	28:
		tbTBLog := CONCAT(tbTBLog, INT_TO_STRING(iTestStep));
		FOR i := 1 TO 3 DO
			IF gaTemps[i].stDescription.xFault = TRUE OR gaTemps[i].stDescription.xAlarm = TRUE THEN
				tbTBLog := CONCAT(tbTBLog, 'F');
				iTestStep := 66;
			ELSE
				tbTBLog := CONCAT(tbTBLog, 'S');
				iTestStep := iTestStep + 1;
			END_IF
		END_FOR
	29:
		tbTBLog := CONCAT(tbTBLog, INT_TO_STRING(iTestStep));
		IF gConductivity.stDescription.xFault = FALSE OR gConductivity.stDescription.xAlarm = FALSE THEN
				tbTBLog := CONCAT(tbTBLog, 'F');
				iTestStep := 66;
		ELSE
				tbTBLog := CONCAT(tbTBLog, 'S');
				iTestStep := iTestStep + 1;
		END_IF
	30:
		tbTBLog := CONCAT(tbTBLog, INT_TO_STRING(iTestStep));
		IF gFlow.stDescription.xFault = TRUE OR gFlow.stDescription.xAlarm = TRUE THEN
				tbTBLog := CONCAT(tbTBLog, 'F ');
				iTestStep := 66;
		ELSE
				tbTBLog := CONCAT(tbTBLog, 'S');
				iTestStep := iTestStep + 1;
		END_IF
	31: (*Max Val Test Cond Should Fault*)
		resetVars();
		tbTBLog := CONCAT(tbTBLog, INT_TO_STRING(iTestStep));
		gaPumps[1].stPumpPower.iRaw := 5;
		gaPumps[2].stPumpPower.iRaw := 5;
		gaTemps[i].stTempRead.iRaw := 5;
		gaTemps[2].stTempRead.iRaw := 5;
		gaTemps[3].stTempRead.iRaw := 5;
		gConductivity.stConductivity.iRaw := 100;
		gFlow.stFlowRate.iRaw := 5;
		UUT();
		tbTBLog := CONCAT(tbTBLog, 'S');
		iTestStep := iTestStep + 1;
	32:
		tbTBLog := CONCAT(tbTBLog, INT_TO_STRING(iTestStep));
		FOR i := 1 TO 2 DO
			IF gaPumps[i].stDescription.xFault = TRUE OR gaPumps[i].stDescription.xAlarm = TRUE THEN
				tbTBLog := CONCAT(tbTBLog, 'F');
				iTestStep := 66;
			ELSE
				tbTBLog := CONCAT(tbTBLog, 'S');
				iTestStep := iTestStep + 1;
			END_IF
		END_FOR

	33:
		tbTBLog := CONCAT(tbTBLog, INT_TO_STRING(iTestStep));
		FOR i := 1 TO 3 DO
			IF gaTemps[i].stDescription.xFault = TRUE OR gaTemps[i].stDescription.xAlarm = TRUE THEN
				tbTBLog := CONCAT(tbTBLog, 'F');
				iTestStep := 66;
			ELSE
				tbTBLog := CONCAT(tbTBLog, 'S');
				iTestStep := iTestStep + 1;
			END_IF
		END_FOR
	34:
		tbTBLog := CONCAT(tbTBLog, INT_TO_STRING(iTestStep));
		IF gConductivity.stDescription.xFault = FALSE OR gConductivity.stDescription.xAlarm = FALSE THEN
				tbTBLog := CONCAT(tbTBLog, 'F');
				iTestStep := 66;
		ELSE
				tbTBLog := CONCAT(tbTBLog, 'S');
				iTestStep := iTestStep + 1;
		END_IF
	35:
		tbTBLog := CONCAT(tbTBLog, INT_TO_STRING(iTestStep));
		IF gFlow.stDescription.xFault = TRUE OR gFlow.stDescription.xAlarm = TRUE THEN
				tbTBLog := CONCAT(tbTBLog, 'F ');
				iTestStep := 66;
		ELSE
				tbTBLog := CONCAT(tbTBLog, 'S');
				iTestStep := iTestStep + 1;
		END_IF
	36: (*MIN Val Test Flow Should Fault*)
		resetVars();
		tbTBLog := CONCAT(tbTBLog, INT_TO_STRING(iTestStep));
		gaPumps[1].stPumpPower.iRaw := 5;
		gaPumps[2].stPumpPower.iRaw := 5;
		gaTemps[i].stTempRead.iRaw := 5;
		gaTemps[2].stTempRead.iRaw := 5;
		gaTemps[3].stTempRead.iRaw := 5;
		gConductivity.stConductivity.iRaw := 5;
		gFlow.stFlowRate.iRaw := 1;
		UUT();
		tbTBLog := CONCAT(tbTBLog, 'S');
		iTestStep := iTestStep + 1;
	37:
		tbTBLog := CONCAT(tbTBLog, INT_TO_STRING(iTestStep));
		FOR i := 1 TO 2 DO
			IF gaPumps[i].stDescription.xFault = TRUE OR gaPumps[i].stDescription.xAlarm = TRUE THEN
				tbTBLog := CONCAT(tbTBLog, 'F');
				iTestStep := 66;
			ELSE
				tbTBLog := CONCAT(tbTBLog, 'S');
				iTestStep := iTestStep + 1;
			END_IF
		END_FOR

	38:
		tbTBLog := CONCAT(tbTBLog, INT_TO_STRING(iTestStep));
		FOR i := 1 TO 3 DO
			IF gaTemps[i].stDescription.xFault = TRUE OR gaTemps[i].stDescription.xAlarm = TRUE THEN
				tbTBLog := CONCAT(tbTBLog, 'F');
				iTestStep := 66;
			ELSE
				tbTBLog := CONCAT(tbTBLog, 'S');
				iTestStep := iTestStep + 1;
			END_IF
		END_FOR
	39:
		tbTBLog := CONCAT(tbTBLog, INT_TO_STRING(iTestStep));
		IF gConductivity.stDescription.xFault = TRUE OR gConductivity.stDescription.xAlarm = TRUE THEN
				tbTBLog := CONCAT(tbTBLog, 'F');
				iTestStep := 66;
		ELSE
				tbTBLog := CONCAT(tbTBLog, 'S');
				iTestStep := iTestStep + 1;
		END_IF
	40:
		tbTBLog := CONCAT(tbTBLog, INT_TO_STRING(iTestStep));
		IF gFlow.stDescription.xFault = FALSE  OR gFlow.stDescription.xAlarm = FALSE THEN
				tbTBLog := CONCAT(tbTBLog, 'F ');
				iTestStep := 66;
		ELSE
				tbTBLog := CONCAT(tbTBLog, 'S');
				iTestStep := iTestStep + 1;
		END_IF
	41: (*MAX Val Test Flow Should Fault*)
		resetVars();
		tbTBLog := CONCAT(tbTBLog, INT_TO_STRING(iTestStep));
		gaPumps[1].stPumpPower.iRaw := 5;
		gaPumps[2].stPumpPower.iRaw := 5;
		gaTemps[i].stTempRead.iRaw := 5;
		gaTemps[2].stTempRead.iRaw := 5;
		gaTemps[3].stTempRead.iRaw := 5;
		gConductivity.stConductivity.iRaw := 5;
		gFlow.stFlowRate.iRaw := 100;
		UUT();
		tbTBLog := CONCAT(tbTBLog, 'S');
		iTestStep := iTestStep + 1;
	42:
		tbTBLog := CONCAT(tbTBLog, INT_TO_STRING(iTestStep));
		FOR i := 1 TO 2 DO
			IF gaPumps[i].stDescription.xFault = TRUE OR gaPumps[i].stDescription.xAlarm = TRUE THEN
				tbTBLog := CONCAT(tbTBLog, 'F');
				iTestStep := 66;
			ELSE
				tbTBLog := CONCAT(tbTBLog, 'S');
				iTestStep := iTestStep + 1;
			END_IF
		END_FOR

	43:
		tbTBLog := CONCAT(tbTBLog, INT_TO_STRING(iTestStep));
		FOR i := 1 TO 3 DO
			IF gaTemps[i].stDescription.xFault = TRUE OR gaTemps[i].stDescription.xAlarm = TRUE THEN
				tbTBLog := CONCAT(tbTBLog, 'F');
				iTestStep := 66;
			ELSE
				tbTBLog := CONCAT(tbTBLog, 'S');
				iTestStep := iTestStep + 1;
			END_IF
		END_FOR
	44:
		tbTBLog := CONCAT(tbTBLog, INT_TO_STRING(iTestStep));
		IF gConductivity.stDescription.xFault = TRUE OR gConductivity.stDescription.xAlarm = TRUE THEN
				tbTBLog := CONCAT(tbTBLog, 'F');
				iTestStep := 66;
		ELSE
				tbTBLog := CONCAT(tbTBLog, 'S');
				iTestStep := iTestStep + 1;
		END_IF
	45:
		tbTBLog := CONCAT(tbTBLog, INT_TO_STRING(iTestStep));
		IF gFlow.stDescription.xFault = FALSE  OR gFlow.stDescription.xAlarm = FALSE THEN
				tbTBLog := CONCAT(tbTBLog, 'F ');
				iTestStep := 66;
		ELSE
				tbTBLog := CONCAT(tbTBLog, 'S');
				iTestStep := iTestStep + 1;
		END_IF
END_CASE
*)
END_PROGRAM

(* POU Legacy/FB_TempValCtrlSys, ST *)
FUNCTION_BLOCK FB_TempValCtrlSys
VAR_INPUT
END_VAR
VAR_OUTPUT
END_VAR
VAR
	tM: ARRAY [1..3] OF REAL; (*Temperature Measuremnts*)
	tD: ARRAY [1..3] OF REAL; (*Temperature differences of 1 and 2, 1 and 3, 2 and 3*)
	tCF: ARRAY [1..3] OF BOOL; (*Candiates of potential temperatures that failed. First true means 1 and 2. Second true means 1 and 3. And third true means 2 and 3.*)
	tCA: ARRAY [1..3] OF BOOL; (*Candiates of potential temperatures that alarmed. First true means 1 and 2. Second true means 1 and 3. And third true means 2 and 3.*)

	i: INT;
	diffThreshold: REAL;
	diffTolerance: REAL;
	faultCount: INT; (*How many faults*)
	sysMeasMode: INT;
END_VAR
faultCount := 0;
i := 0;
(*Subtract to find differneces between temperatures*)
FOR i := 1 TO 3 DO
	tM[i] := gaTemps[i].stTempRead.rProcessed;
END_FOR
tD[1] := ABS(tM[1] - tM[2]);
tD[2] := ABS(tM[1] - tM[3]);
tD[3] := ABS(tM[2] - tM[3]);
i := 0;
FOR i := 1 TO 3 DO
	IF tD[i] > gTempValCtrlSys.rDiffThresh THEN
		tCF[i] := TRUE;
		tCA[i] := TRUE;
		faultCount := faultCount + 1;
		gTempValCtrlSys.xAlarm := TRUE;
	ELSIF tD[i] > (gTempValCtrlSys.rDiffTol) THEN
		tCA[i] := TRUE;
		gTempValCtrlSys.xAlarm := TRUE;
END_IF
END_FOR
IF tCF[1] = TRUE AND tCF[2] = TRUE AND tCF[3] = TRUE THEN
	FOR i := 1 TO 3 DO
		gaTemps[i].stDescription.xFault := TRUE;
	END_FOR
ELSIF tCF[1] = TRUE AND tCF[2] = TRUE AND tCF[3] = FALSE THEN
	gaTemps[1].stDescription.xFault := TRUE;
ELSIF tCF[1] = TRUE AND tCF[2] = FALSE AND tCF[3] = TRUE THEN
	gaTemps[2].stDescription.xFault := TRUE;
ELSIF tCF[1] = FALSE AND tCF[2] = TRUE AND tCF[3] = TRUE THEN
	gaTemps[3].stDescription.xFault := TRUE;

END_IF

IF tCA[1] = TRUE AND tCA[2] = TRUE AND tCA[3] = TRUE THEN
	FOR i := 1 TO 3 DO
		gaTemps[i].stDescription.xAlarm:= TRUE;
	END_FOR
ELSIF tCA[1] = TRUE AND tCA[2] = TRUE AND tCA[3] = FALSE THEN
	gaTemps[1].stDescription.xAlarm := TRUE;
ELSIF tCA[1] = TRUE AND tCA[2] = FALSE AND tCA[3] = TRUE THEN
	gaTemps[2].stDescription.xAlarm := TRUE;
ELSIF tCA[1] = FALSE AND tCA[2] = TRUE AND tCA[3] = TRUE THEN
	gaTemps[3].stDescription.xAlarm := TRUE;
END_IF

IF faultCount = 0 THEN
	sysMeasMode := 0;
ELSIF faultCount = 1 THEN
	gProgramErrors.xTempValCtrlSys  := TRUE; (*If difference between only two RTDs off, means poor values selected*)
	gTempValCtrlSys.xFault := TRUE;
	gTempValCtrlSys.xAlarm := TRUE;
ELSIF faultCount = 2 THEN (*Means that an RTD failed, will need to take average *)
	sysMeasMode := 1;
	gTempValCtrlSys.xAlarm := TRUE;
ELSIF faultCount = 3 THEN (*All RTDs failed, system fault*)
	sysMeasMode := 2;
	gTempValCtrlSys.xFault := TRUE;
	gTempValCtrlSys.xAlarm := TRUE;
ELSE (*Should not happen*)
	gProgramErrors.xTempValCtrlSys  := TRUE;
	gTempValCtrlSys.xFault := TRUE;
	gTempValCtrlSys.xAlarm := TRUE;
END_IF
END_FUNCTION_BLOCK

(* POU Test Bench Folder/TB_VALIDATE, LD *)
PROGRAM TB_VALIDATE
VAR
	rResult: REAL;
	rinput: REAL;
	rMax: REAL;
	rMin: REAL;
	Val1: REAL;
	Val2: REAL;
	Val3: REAL;
	bool1: BOOL := TRUE;
	bool2: BOOL := TRUE;
	bool3: BOOL := TRUE;
END_VAR
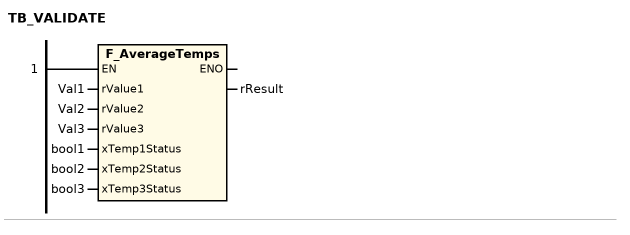
_LD_ (* Ladder Diagram *)
NETWORK 1
	*
		EN --- F_AverageTemps(rValue1: Val1, rValue2: Val2, rValue3: Val3, xTemp1Status: bool1, xTemp2Status: bool2, xTemp3Status: bool3) => rResult
_END_LD_
(* the same logic as Structured Text *)
(* Network 1 *)
rResult := F_AverageTemps(rValue1 := Val1, rValue2 := Val2, rValue3 := Val3, xTemp1Status := bool1, xTemp2Status := bool2, xTemp3Status := bool3);
END_PROGRAM

(* POU Test Bench Folder/TB_WaterLevelCheck, LD *)
PROGRAM TB_WaterLevelCheck
VAR
	fbcwl: FB_CheckWaterLevel;
	sys: ST_SYSTEM;
	wl: BOOL := FALSE;
	wll: BOOL := FALSE;
	flags: ST_InstrumentFlags;
END_VAR
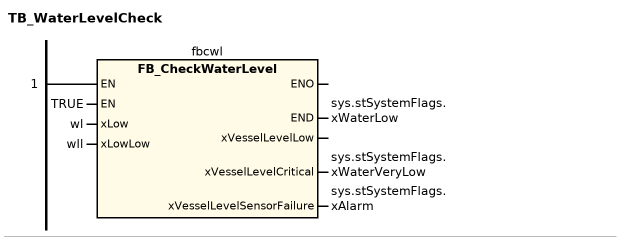
_LD_ (* Ladder Diagram *)
NETWORK 1
	*
		EN --- fbcwl:FB_CheckWaterLevel(EN: TRUE, xLow: wl, xLowLow: wll, xVesselLevelCritical => sys.stSystemFlags.xWaterVeryLow, xVesselLevelSensorFailure => sys.stSystemFlags.xAlarm) => sys.stSystemFlags.xWaterLow
_END_LD_
(* the same logic as Structured Text *)
(* Network 1 *)
fbcwl(EN := TRUE, xLow := wl, xLowLow := wll);
sys.stSystemFlags.xWaterVeryLow := fbcwl.xVesselLevelCritical;
sys.stSystemFlags.xAlarm := fbcwl.xVesselLevelSensorFailure;
sys.stSystemFlags.xWaterLow := fbcwl.END;
END_PROGRAM

(* POU System Startup/F_InitSystemCheck, ST *)
FUNCTION F_InitSystemCheck : BOOL
VAR_INPUT
	xSystemRunSwitch: BOOL;
	xSystemFaultFlag: BOOL;
END_VAR
VAR
END_VAR
IF (xSystemRunSwitch AND xSystemFaultFlag) OR (xSystemRunSwitch = FALSE) THEN
	F_InitSystemCheck := FALSE;
ELSIF xSystemRunSwitch AND xSystemFaultFlag = FALSE THEN
	F_InitSystemCheck := TRUE;
END_IF;
END_FUNCTION

(* POU Instrument Control/F_SystemFaultCheck, LD *)
FUNCTION_BLOCK F_SystemFaultCheck
VAR_INPUT
	xRTD1: BOOL;
	xRTD2: BOOL;
	xRTD3: BOOL;
	xPump1: BOOL;
	xBadWaterLevelSensor: BOOL;
	xBadConductivitySensor: BOOL;
	xBadFlowSensor: BOOL;
	xBadTemperature: BOOL;
	xLowPressure: BOOL;
	xLowFLow: BOOL;
	xNoBackup: BOOL;
	iActivePump: INT;
	xBadActuate: BOOL;
	xSystemPump1Activate: BOOL;
	xSystemPump2Activate: BOOL;
END_VAR
VAR_OUTPUT
	xSystemFault: BOOL;
END_VAR
VAR
	xBadTemp12: BOOL;
	xBadTemp23: BOOL;
	xBadTemp31: BOOL;
	xPump2: BOOL;
	xNoPump: BOOL;
	xTri1: BOOL;
	xTri2: BOOL;
	xTri3: BOOL;
END_VAR
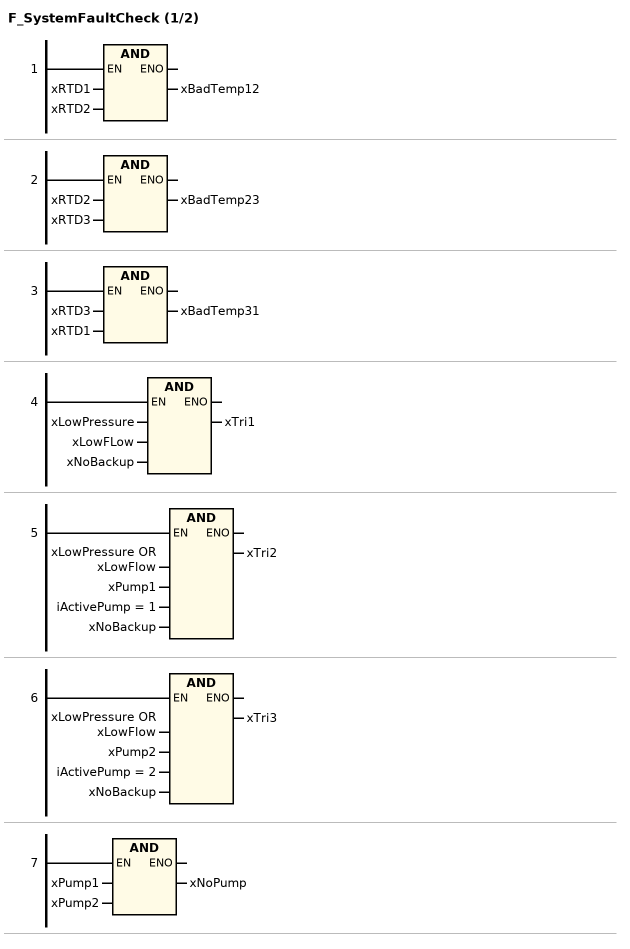
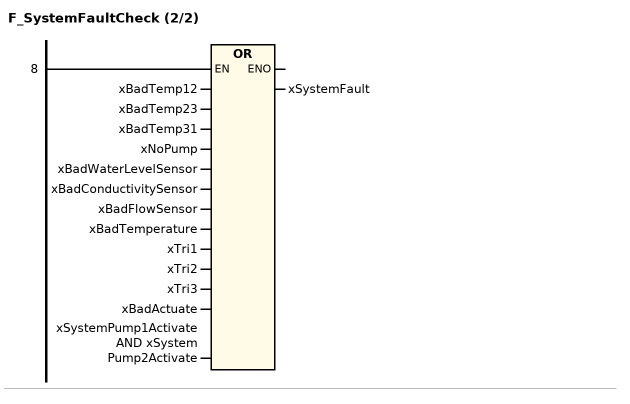
_LD_ (* Ladder Diagram *)
NETWORK 1
	*
		EN --- AND(xRTD1, xRTD2) => xBadTemp12
NETWORK 2
	*
		EN --- AND(xRTD2, xRTD3) => xBadTemp23
NETWORK 3
	*
		EN --- AND(xRTD3, xRTD1) => xBadTemp31
NETWORK 4
	*
		EN --- AND(xLowPressure, xLowFLow, xNoBackup) => xTri1
NETWORK 5
	*
		EN --- AND(xLowPressure OR xLowFlow, xPump1, iActivePump = 1, xNoBackup) => xTri2
NETWORK 6
	*
		EN --- AND(xLowPressure OR xLowFlow, xPump2, iActivePump = 2, xNoBackup) => xTri3
NETWORK 7
	*
		EN --- AND(xPump1, xPump2) => xNoPump
NETWORK 8
	*
		EN --- OR(xBadTemp12, xBadTemp23, xBadTemp31, xNoPump, xBadWaterLevelSensor, xBadConductivitySensor, xBadFlowSensor, xBadTemperature, xTri1, xTri2, xTri3, xBadActuate, xSystemPump1Activate AND xSystemPump2Activate) => xSystemFault
_END_LD_
(* the same logic as Structured Text *)
(* Network 1 *)
xBadTemp12 := xRTD1 AND xRTD2;
(* Network 2 *)
xBadTemp23 := xRTD2 AND xRTD3;
(* Network 3 *)
xBadTemp31 := xRTD3 AND xRTD1;
(* Network 4 *)
xTri1 := xLowPressure AND xLowFLow AND xNoBackup;
(* Network 5 *)
xTri2 := (xLowPressure OR xLowFlow) AND xPump1 AND (iActivePump = 1) AND xNoBackup;
(* Network 6 *)
xTri3 := (xLowPressure OR xLowFlow) AND xPump2 AND (iActivePump = 2) AND xNoBackup;
(* Network 7 *)
xNoPump := xPump1 AND xPump2;
(* Network 8 *)
xSystemFault := xBadTemp12 OR xBadTemp23 OR xBadTemp31 OR xNoPump OR xBadWaterLevelSensor OR xBadConductivitySensor OR xBadFlowSensor OR xBadTemperature OR xTri1 OR xTri2 OR xTri3 OR xBadActuate OR (xSystemPump1Activate AND xSystemPump2Activate);
END_FUNCTION_BLOCK

(* POU Instrument Control/Temperature Control/F_TemperatureController, ST *)
FUNCTION F_TemperatureController : REAL
VAR_INPUT
	xSystemFaultFlag: BOOL;
	xAwaitInit: BOOL;
	rTemperatureInput: REAL;
	rSetpoint: REAL;
END_VAR
VAR
	rOutput: REAL;
END_VAR
IF xSystemFaultFlag OR xAwaitInit THEN
	F_TemperatureController := 1;
ELSE
	F_TemperatureController :=( rTemperatureInput/2)/rTemperatureInput;
END_IF
END_FUNCTION

(* POU Functions/F_ValueCap, ST *)
FUNCTION F_ValueCap : REAL
VAR_INPUT
	rInput: REAL;
END_VAR
VAR
END_VAR
IF (rInput > 1) THEN
	F_ValueCap := 1;
ELSIF (rInput < 1) THEN
	F_ValueCap := 0;
ELSE
	F_ValueCap := rInput;
END_IF
END_FUNCTION

(* POU Data Conversion/System -> Instrument/FB_ActivePumpSet, ST *)
FUNCTION_BLOCK FB_ActivePumpSet
VAR_INPUT
	xSystemPump1Actuate: BOOL;
	xSystemPump2Actuate: BOOL;
END_VAR
VAR_OUTPUT
	iActivePump: INT;
	xSystemFaultFlag: BOOL;
END_VAR
VAR
END_VAR
IF xSystemPump1Actuate AND xSystemPump2Actuate = FALSE THEN
	iActivePump := 1;
ELSIF xSystemPump2Actuate AND xSystemPump1Actuate = FALSE THEN
	iActivePump := 2;
ELSIF xSystemPump1Actuate AND xSystemPump2Actuate THEN
	iActivePump := 0;
	xSystemFaultFlag := TRUE;
ELSIF xSystemPump1Actuate = FALSE AND xSystemPump2Actuate = FALSE THEN
	iActivePump := 0;
END_IF
END_FUNCTION_BLOCK

(* POU Data Conversion/Instrument -> Signal/FB_ActuateAnalog, LD *)
 FUNCTION_BLOCK FB_ActuateAnalog
VAR_INPUT
	rActuateValue: REAL;
END_VAR
VAR_OUTPUT
	wActuateSignal: WORD;
END_VAR
VAR
	rScaledValue: REAL;
END_VAR
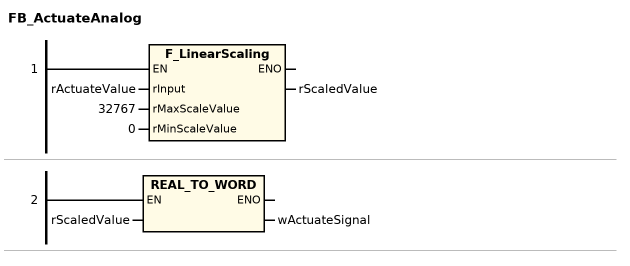
_LD_ (* Ladder Diagram *)
NETWORK 1
	*
		EN --- F_LinearScaling(rInput: rActuateValue, rMaxScaleValue: 32767, rMinScaleValue: 0) => rScaledValue
NETWORK 2
	*
		EN --- REAL_TO_WORD(rScaledValue) => wActuateSignal
_END_LD_
(* the same logic as Structured Text *)
(* Network 1 *)
rScaledValue := F_LinearScaling(rInput := rActuateValue, rMaxScaleValue := 32767, rMinScaleValue := 0);
(* Network 2 *)
wActuateSignal := REAL_TO_WORD(rScaledValue);
END_FUNCTION_BLOCK

(* POU Data Conversion/Instrument -> Signal/FB_ActuateDigital, LD *)
FUNCTION_BLOCK FB_ActuateDigital
VAR_INPUT
	xPump1ActuateValue: BOOL;
	xPump2ActuateValue: BOOL;
	xFan12ActuateValue: BOOL;
	xFan34ActuateValue: BOOL;
END_VAR
VAR_OUTPUT
	xPump1OutputSignal: BOOL;
	xPump2OutputSignal: BOOL;
	xFan12OutputSignal: BOOL;
	xFan34OutputSignal: BOOL;
END_VAR
VAR
END_VAR
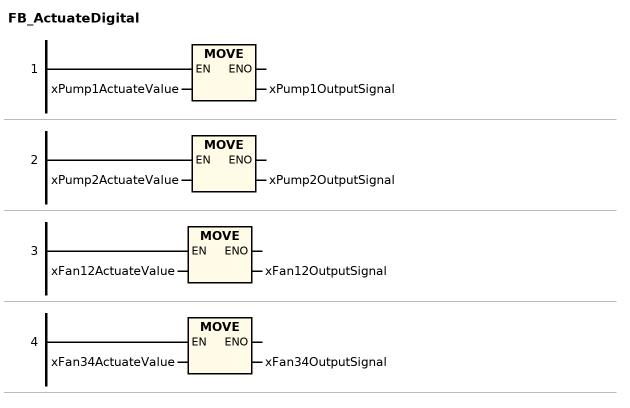
_LD_ (* Ladder Diagram *)
NETWORK 1
	*
		EN --- MOVE(xPump1ActuateValue) => xPump1OutputSignal
NETWORK 2
	*
		EN --- MOVE(xPump2ActuateValue) => xPump2OutputSignal
NETWORK 3
	*
		EN --- MOVE(xFan12ActuateValue) => xFan12OutputSignal
NETWORK 4
	*
		EN --- MOVE(xFan34ActuateValue) => xFan34OutputSignal
_END_LD_
(* the same logic as Structured Text *)
(* Network 1 *)
xPump1OutputSignal := xPump1ActuateValue;
(* Network 2 *)
xPump2OutputSignal := xPump2ActuateValue;
(* Network 3 *)
xFan12OutputSignal := xFan12ActuateValue;
(* Network 4 *)
xFan34OutputSignal := xFan34ActuateValue;
END_FUNCTION_BLOCK

(* POU Data Conversion/System -> Instrument/FB_ActuateFilter, ST *)
FUNCTION_BLOCK FB_ActuateFilter
VAR_INPUT
	rActuateValue: REAL;
	rActuateMAX: REAL;
	rActuateMIN: REAL;
END_VAR
VAR_OUTPUT
	rOutput: REAL;
END_VAR
VAR
	xBadActuateValue: BOOL;
	rLastReadValue: REAL;
END_VAR
IF rActuateValue > rActuateMAX OR rActuateValue < rActuateMIN THEN
	xBadActuateValue := TRUE;
	rOutput := rLastReadValue;
ELSIF rActuateValue > 1 THEN
	rLastReadValue := rOutput;
	rOutput := 1;
ELSIF rActuateValue < 0 THEN
	rLastReadValue := rOutput;
	rOutput := 0;
ELSE
	rLastReadValue := rOutput;
	rOutput := rActuateValue;
END_IF
END_FUNCTION_BLOCK

(* POU Legacy/FB_AnalogHeartbeatCheck, ST *)
FUNCTION_BLOCK FB_AnalogHeartbeatCheck (*Checks if analog devices are being read*)
VAR
	i: INT;
 a: INT;
END_VAR
VAR_INPUT
	iMinRawThreshold: INT;
	iMaxRawThreshold: INT;
END_VAR
VAR_OUTPUT
END_VAR
FOR i := 1 TO 2 DO
	IF (gaPumps[i].stPumpPower.iRaw < iMinRawThreshold OR gaPumps[i].stPumpPower.iRaw > iMaxRawThreshold)   THEN
		gaPumps[i].stDescription.xAlarm:= TRUE;
		gaPumps[i].stDescription.xFault:= TRUE;
	END_IF
END_FOR
FOR i := 1 TO 3 DO
	IF (gaTemps[i].stTempRead.iRaw < iMinRawThreshold OR gaTemps[i].stTempRead.iRaw > iMaxRawThreshold)  THEN
		gaTemps[i].stDescription.xAlarm:= TRUE;
		gaTemps[i].stDescription.xFault:= TRUE;
	END_IF
END_FOR

IF gConductivity.stConductivity.iRaw < iMinRawThreshold OR gConductivity.stConductivity.iRaw > iMaxRawThreshold THEN
	gConductivity.stDescription.xAlarm := TRUE;
	gConductivity.stDescription.xFault := TRUE;
END_IF

IF gFlow.stFlowRate.iRaw< iMinRawThreshold OR  gFlow.stFlowRate.iRaw > iMaxRawThreshold THEN
	gFlow.stDescription.xAlarm:= TRUE;
	gFlow.stDescription.xFault:= TRUE;
END_IF
END_FUNCTION_BLOCK

(* POU Instrument Checking Functions/FB_BoundCheck, ST *)
FUNCTION_BLOCK FB_BoundCheck
VAR_INPUT
	xEnable: BOOL;
	rInput: REAL;
	xMaxCheck: BOOL;
	xMinCheck: BOOL;
	rMaxVariable: REAL;
	rMinVariable: REAL;
	rTolerance: REAL;
END_VAR
VAR_OUTPUT
	xDone: BOOL;
	xPastBoundFlag: BOOL;
END_VAR
VAR
END_VAR
IF xEnable = FALSE  THEN
	RETURN;
END_IF;
IF xMaxCheck = TRUE AND xMinCheck = TRUE THEN
	IF rInput > (rMaxVariable + rTolerance) THEN
		xPastBoundFlag := TRUE;
	ELSIF rInput < (rMinVariable - rTolerance) THEN
		xPastBoundFlag := TRUE;
	END_IF
ELSIF xMaxCheck = TRUE THEN
	IF rInput > (rMaxVariable + rTolerance) THEN
		xPastBoundFlag := TRUE;
	END_IF
ELSIF xMinCheck = TRUE THEN
	IF rInput < (rMinVariable - rTolerance) THEN
		xPastBoundFlag := TRUE;
	END_IF
END_IF


xDone := TRUE;
(*Validated 3/9/26*)
END_FUNCTION_BLOCK

(* POU Instrument Control/FB_FanActuation, ST *)
FUNCTION_BLOCK FB_FanActuation
VAR_INPUT
	xFanGroup1ON: BOOL;
	xFanGroup2ON: BOOL;
END_VAR
VAR_OUTPUT
	xFan12Actuate: BOOL := TRUE;
END_VAR
VAR
	xFan23Actuate: BOOL := FALSE;
END_VAR
IF xFanGroup1ON = FALSE  THEN
	xFan12Actuate := FALSE;
ELSE
	xFan12Actuate := TRUE;
END_IF
IF xFanGroup2ON = TRUE THEN
	xFan23Actuate := TRUE;
ELSE
	xFan23Actuate := FALSE;
END_IF
END_FUNCTION_BLOCK

(* POU Instrument Control/Check Control/FB_InitializationTimer, ST *)
FUNCTION_BLOCK FB_InitializationTimer
VAR_INPUT
	tInitTime: TIME;
END_VAR
VAR_OUTPUT
END_VAR
VAR
	fbTimerOn: TON;
	xInit: BOOL;
END_VAR
VAR_IN_OUT
	xAwaitInit: BOOL;
END_VAR
IF xAwaitInit AND xInit = FALSE THEN
	xInit := TRUE;
END_IF

fbTimerOn(IN := xInit, PT := tInitTime);

IF fbTimerOn.Q = TRUE THEN
	xAwaitInit := FALSE;
	xInit := FALSE;
END_IF
END_FUNCTION_BLOCK

(* POU System Startup/FB_InitSystemCheck, ST *)
FUNCTION_BLOCK FB_InitSystemCheck
VAR_INPUT
	xSystemRunSwitch: BOOL;
	xSystemFaultFlag: BOOL;
END_VAR
VAR_OUTPUT
	xExecute: BOOL;
END_VAR
VAR
END_VAR
IF (xSystemRunSwitch AND xSystemFaultFlag) OR (xSystemRunSwitch = FALSE) THEN
	RETURN;
ELSIF xSystemRunSwitch AND xSystemFaultFlag = FALSE THEN
	xExecute := TRUE;
END_IF;
END_FUNCTION_BLOCK

(* POU Data Conversion/System -> Instrument/FB_InstrumentSystemAlignment, LD *)
FUNCTION_BLOCK FB_InstrumentSystemAlignment
VAR_INPUT
	xSystemPump1Activate: BOOL;
	xSystemPump2Activate: BOOL;
	xSystemFan12Activate: BOOL;
	xSystemFan34Activate: BOOL;
END_VAR
VAR_OUTPUT
	xPump1Activate: BOOL;
	xPump2Activate: BOOL;
	xFan12Activate: BOOL;
	xFan34Activate: BOOL;
	xSystemFaultFlag: BOOL;
	iActivePump: INT;
END_VAR
VAR
	fbactivepumpset: FB_ActivePumpSet;
END_VAR
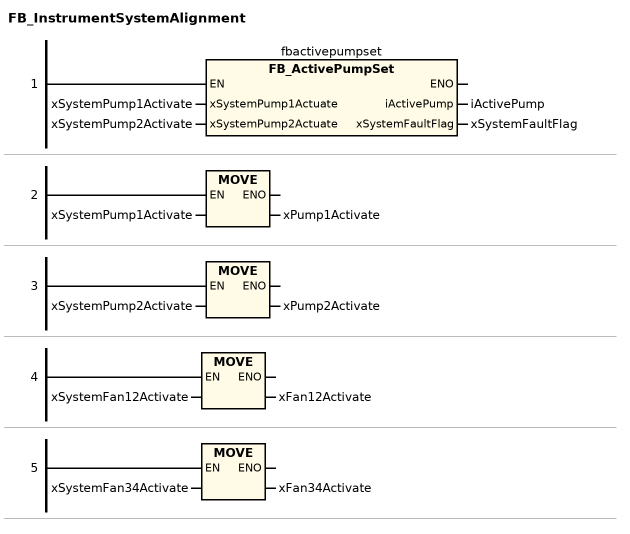
_LD_ (* Ladder Diagram *)
NETWORK 1
	*
		EN --- fbactivepumpset:FB_ActivePumpSet(xSystemPump1Actuate: xSystemPump1Activate, xSystemPump2Actuate: xSystemPump2Activate, xSystemFaultFlag => xSystemFaultFlag) => iActivePump
NETWORK 2
	*
		EN --- MOVE(xSystemPump1Activate) => xPump1Activate
NETWORK 3
	*
		EN --- MOVE(xSystemPump2Activate) => xPump2Activate
NETWORK 4
	*
		EN --- MOVE(xSystemFan12Activate) => xFan12Activate
NETWORK 5
	*
		EN --- MOVE(xSystemFan34Activate) => xFan34Activate
_END_LD_
(* the same logic as Structured Text *)
(* Network 1 *)
fbactivepumpset(xSystemPump1Actuate := xSystemPump1Activate, xSystemPump2Actuate := xSystemPump2Activate);
xSystemFaultFlag := fbactivepumpset.xSystemFaultFlag;
iActivePump := fbactivepumpset.iActivePump;
(* Network 2 *)
xPump1Activate := xSystemPump1Activate;
(* Network 3 *)
xPump2Activate := xSystemPump2Activate;
(* Network 4 *)
xFan12Activate := xSystemFan12Activate;
(* Network 5 *)
xFan34Activate := xSystemFan34Activate;
END_FUNCTION_BLOCK

(* POU Instrument Control/FB_PumpLogic, ST *)
FUNCTION_BLOCK FB_PumpLogic
VAR_INPUT
	EN: BOOL;
	xPPFE: BOOL;
	xPumpError: BOOL;
	xPrimaryPumpError: BOOL;
	xPrimaryPumpActive: BOOL;
	xSecondaryPumpError: BOOL;
	xSecondaryPumpActive: BOOL;

END_VAR
VAR_OUTPUT
	END: BOOL;
	xAutoHandover: BOOL;
	xPumpFault: BOOL;
END_VAR
VAR
END_VAR
VAR_IN_OUT
	xSimplexPump: BOOL;
END_VAR
END := FALSE;
IF EN = FALSE THEN
	RETURN;
END_IF


IF xSimplexPump = FALSE AND (xPPFE OR (xPrimaryPumpError AND xPrimaryPumpActive) OR (xSecondaryPumpError AND xSecondaryPumpActive)) THEN
	xSimplexPump := TRUE;
	xAutoHandover := TRUE;
ELSIF xSimplexPump = TRUE AND (xPPFE OR (xPrimaryPumpError AND xPrimaryPumpActive) OR (xSecondaryPumpError AND xSecondaryPumpActive)) THEN
	xPumpFault := TRUE;
	xAutoHandover := FALSE;
ELSE
	xAutoHandover := FALSE;
END_IF
END_FUNCTION_BLOCK

(* POU FB_PumpValueSelection, ST *)
FUNCTION_BLOCK FB_PumpValueSelection
VAR_INPUT
	EN: BOOL;
	xPoorReadPrimary: BOOL;
	xPoorReadSecondary: BOOL;
	xPrimaryPumpActive: BOOL;
	xSecondaryPumpActive: BOOL;
END_VAR
VAR_OUTPUT
	END: BOOL;
	xRequestPumpTurnover: BOOL;
END_VAR
VAR
END_VAR
END := FALSE;
IF EN = FALSE THEN
	RETURN;
END_IF

IF (xPoorReadPrimary AND xPrimaryPumpActive) OR (xPoorReadSecondary AND xSecondaryPumpActive) THEN
	xRequestPumpTurnover := TRUE;
ELSE
	xRequestPumpTurnover := FALSE;
END_IF
END := TRUE;
END_FUNCTION_BLOCK

(* POU Instrument Control/FB_SystemAlarmCheck, ST *)
FUNCTION_BLOCK FB_SystemAlarmCheck
VAR_INPUT
	xBadTemp1: BOOL;
	xBadTemp2: BOOL;
	xBadTemp3: BOOL;
	xBadPump1: BOOL;
	xBadPump2: BOOL;
	xBadPumpPower1: BOOL;
	xBadPumpPower2: BOOL;
	xLowPres: BOOL;
	xLowFlow: BOOL;
	xLowWater: BOOL;
	xVeryLowWater: BOOL;
	xBadTemp: BOOL;
	xConductivityAlarm: BOOL;
	xSystemFaultFlag: BOOL;
END_VAR
VAR_OUTPUT
	xSystemAlarmFlag: BOOL;
END_VAR
VAR
	xBadTempSense: BOOL;
	xBadPump: BOOL;
	xBadTri: BOOL;
	xLW: BOOL;
END_VAR
xLW := xLowWater OR xVeryLowWater;
xBadTri := xLowPres OR xLowFlow;
xBadPump := xBadPump1 OR xBadPump2 OR xBadPumpPower1 OR xBadPumpPower2;
xBadTempSense := xBadTemp1 OR xBadTemp2 OR xBadTemp3;
IF xSystemFaultFlag OR xLW OR xBadTri OR xBadPump OR xBadTempSense OR xBadTemp OR xConductivityAlarm THEN
	xSystemAlarmFlag := TRUE;
ELSE
	xSystemAlarmFlag := FALSE;
END_IF
END_FUNCTION_BLOCK

(* POU System Startup/FB_SystemInit, ST *)
FUNCTION_BLOCK FB_SystemInit
VAR_INPUT
	xExecute: BOOL;

END_VAR
VAR_OUTPUT
	xSystemOnFlag: BOOL;
	xFanGroup1Activate: BOOL;
	xPump1Activate: BOOL;
	xAwaitInit: BOOL;
	iActivePump: INT;
END_VAR
VAR
END_VAR
IF xExecute = FALSE THEN
	RETURN;
ELSE
	xFanGroup1Activate := TRUE;
	xPump1Activate := TRUE;
	iActivePump := 1;
	xAwaitInit := TRUE;
	xSystemOnFlag := TRUE;
END_IF;
END_FUNCTION_BLOCK

(* POU Instrument Control/FB_SystemShutdownProcedure, ST *)
FUNCTION_BLOCK FB_SystemShutdownProcedure
VAR_INPUT
	xSystemFaultFlag: BOOL;

END_VAR
VAR_OUTPUT
	xSystemPump1Activate: BOOL;
	xSystemPump2Activate: BOOL;
	xSystemFan12Activate: BOOL;
	xSystemFan34Activate: BOOL;
	xSystemFaultActivate: BOOL;
	xSystemAlarmActivate: BOOL;
	xSystemShutdown: BOOL;
	rValveBypass: REAL;
END_VAR
VAR

END_VAR
IF xSystemFaultFlag OR xSystemShutdown THEN
	xSystemPump1Activate := FALSE;
	xSystemPump2Activate := FALSE;
	xSystemFan12Activate := FALSE;
	xSystemFan34Activate := FALSE;
	xSystemFaultActivate := TRUE;
	xSystemAlarmActivate := TRUE;
	rValveBypass := 0;
	xSystemShutdown := TRUE;
END_IF
END_FUNCTION_BLOCK

(* POU Legacy/FB_tbTempValFuncCheck, ST *)
FUNCTION_BLOCK FB_tbTempValFuncCheck
VAR_INPUT
		aExpectedFaultStatus: ARRAY [1..3] OF BOOL;
		aExpectedAlarmStatus: ARRAY[1..3] OF BOOL;
		xExpectedCtrlSysFault: BOOL;
		xExpectedCtrlSysAlarm: BOOL;
		iExpectediSysMeasState: INT;
END_VAR
VAR_OUTPUT
	xFail: BOOL;
	xSucess: BOOL;
	sState: STRING := 'C';
END_VAR
VAR
	i: INT;
	iCheckStep: INT := 0;
END_VAR
CASE iCheckStep OF
	0:
		CONCAT(sState, INT_TO_STRING(iCheckStep));
		FOR i := 1 TO 3 DO
			IF aExpectedFaultStatus[i] <> gaTemps[i].stDescription.xFault THEN
				xFail := TRUE;
				CONCAT(sState, 'F');
			ELSE
				CONCAT(sState, 'S');
			END_IF
		END_FOR
		iCheckStep := iCheckStep + 1;
	1:
		CONCAT(sState, INT_TO_STRING(iCheckStep));
		FOR i := 1 TO 3 DO
			IF aExpectedAlarmStatus[i] <> gaTemps[i].stDescription.xAlarm THEN
				xFail := TRUE;
				CONCAT(sState, 'F');
			ELSE
				CONCAT(sState, 'S');
			END_IF
		END_FOR
		iCheckStep := iCheckStep + 1;
	2:
		CONCAT(sState, INT_TO_STRING(iCheckStep));
		IF gTempValCtrlSys.xFault <> xExpectedCtrlSysFault THEN
			xFail := TRUE;
			CONCAT(sState, 'F');
		ELSE
			CONCAT(sState, 'S');
		END_IF
		iCheckStep := iCheckStep + 1;
	3:
		CONCAT(sState, INT_TO_STRING(iCheckStep));
		IF gTempValCtrlSys.iSysMeasState <> iExpectediSysMeasState THEN
			xFail := TRUE;
			CONCAT(sState, 'F');
		ELSE
			CONCAT(sState, 'S');
		END_IF
		iCheckStep := iCheckStep + 1;
	4:
		CONCAT(sState, INT_TO_STRING(iCheckStep));
		IF xFail = FALSE THEN
			xSucess := TRUE;
			CONCAT(sState, 'S');
		ELSE
			CONCAT(sState, 'F');
		END_IF


END_CASE
END_FUNCTION_BLOCK

(* POU Legacy/FB_tbTempValFuncSet, ST *)
FUNCTION_BLOCK FB_tbTempValFuncSet
VAR_INPUT
	rSetTemp: ARRAY [1..3] OF REAL;
	iSetState: INT;
	rSetThresh: REAL;
	rSetTol: REAL;
	xTempFault: ARRAY [1..3] OF BOOL;
	xTempAlarm: ARRAY [1..3] OF BOOL;
	xCtrlSysFault: BOOL;
	xCtrlSysAlarm: BOOL;
END_VAR
VAR_OUTPUT
END_VAR
VAR
	i: INT;
END_VAR
FOR i := 1 TO 3 DO
	gaTemps[i].stTempRead.rProcessed := rSetTemp[i];
	gaTemps[i].stDescription.xFault := xTempFault[i];
	gaTemps[i].stDescription.xAlarm := xTempAlarm[i];
END_FOR
gTempValCtrlSys.iSysMeasState := iSetState;
gTempValCtrlSys.rDiffThresh := rSetThresh;
gTempValCtrlSys.rDiffTol:= rSetTol;
gTempValCtrlSys.xAlarm := xCtrlSysFault;
gTempValCtrlSys.xFault := xCtrlSysAlarm;
END_FUNCTION_BLOCK

(* POU Legacy/FB_TempValCS, ST *)
FUNCTION_BLOCK FB_TempValCS
VAR_INPUT
END_VAR
VAR_OUTPUT
END_VAR
VAR
	a: INT;
END_VAR
a := 0;
END_FUNCTION_BLOCK

(* POU Test Bench Folder/TB_FLICKER, ST *)
FUNCTION_BLOCK TB_FLICKER
VAR_INPUT
	xEnable: BOOL;
	xContinouslyBounce: BOOL;
	iBounceCounterLimit: INT;
	iCycleCounterLimit: INT;
	xFinalValue: BOOL;
END_VAR
VAR_OUTPUT
END_VAR
VAR
	fbMetronome: TON;
	iBounceCounter: INT;
	iCycleCounter: INT := 0;
END_VAR

VAR_IN_OUT
	xSimulatedRawInput: BOOL;
END_VAR
IF xEnable = FALSE THEN
	RETURN;
END_IF
(* 1. The Metronome *)
(* By putting 'NOT fbMetronome.Q' into its own input, it automatically 
   restarts itself every 10 milliseconds! *)

iCycleCounter := iCycleCounter + 1;


(* 2. The Flipper *)
(* Every time the timer finishes its 10ms tick... *)

IF iCycleCounter >= iCycleCounterLimit THEN
    
    (* If we haven't bounced 10 times yet, keep flipping the signal ON and OFF *)

	IF xContinouslyBounce = FALSE AND  iBounceCounter < iBounceCounterLimit THEN

		xSimulatedRawInput := NOT xSimulatedRawInput; (* Toggle the boolean *)

		iBounceCounter := iBounceCounter + 1;
        

	ELSIF xContinouslyBounce = FALSE AND iBounceCounter >= iBounceCounterLimit THEN       (* After 10 bounces, hold the signal solid TRUE to see if your Debounce catches it *)

		xSimulatedRawInput := xFinalValue; 

	ELSIF xContinouslyBounce = TRUE THEN
		xSimulatedRawInput := NOT xSimulatedRawInput;
	END_IF
    

	iCycleCounter := 0;
END_IF
END_FUNCTION_BLOCK

(* POU Test Bench Folder/TB_HOLDUP, ST *)
FUNCTION_BLOCK TB_HOLDUP
VAR_INPUT
	xEnable: BOOL;
END_VAR
VAR_OUTPUT
END_VAR
VAR
	xWait: BOOL := TRUE;
END_VAR
IF xEnable = FALSE THEN
	RETURN;
END_IF
WHILE xWait DO
	xWait := TRUE;
END_WHILE
END_FUNCTION_BLOCK

(* POU Test Bench Folder/TB_INSTRUMENTRESET, ST *)
FUNCTION_BLOCK TB_INSTRUMENTRESET
VAR_INPUT
	xEnable: BOOL;
END_VAR
VAR_OUTPUT
END_VAR
VAR
END_VAR
VAR_IN_OUT
	stInstrument: ST_INSTRUMENT;
END_VAR
IF xEnable = FALSE THEN
	RETURN;
END_IF
END_FUNCTION_BLOCK

(* POU Test Bench Folder/TB_SET_BOOL, ST *)
FUNCTION_BLOCK TB_SET_BOOL
VAR_INPUT
	xEnable: BOOL;
	xCheck: BOOL;
	newOrCheckValue: BOOL;
END_VAR
VAR_OUTPUT
	xContinue: BOOL := TRUE;
	xTestFailure: BOOL;
END_VAR
VAR_IN_OUT
	oldValue: BOOL;
END_VAR
VAR
END_VAR
IF xEnable = FALSE THEN
	RETURN;
END_IF
IF xCheck = FALSE THEN
	oldValue := newOrCheckValue;
ELSE
	IF oldValue <> newOrCheckValue THEN
		xTestFailure := TRUE;
	END_IF
END_IF
END_FUNCTION_BLOCK

(* POU Test Bench Folder/TB_SET_INT, ST *)
FUNCTION_BLOCK TB_SET_INT
VAR_INPUT
	xEnable: BOOL;
	xCheck: BOOL;
	newOrCheckValue: INT;
END_VAR
VAR_OUTPUT
	xContinue: BOOL := TRUE;
	xTestFailure: BOOL;
END_VAR
VAR_IN_OUT
	oldValue: INT;
END_VAR
VAR
END_VAR
IF xEnable = FALSE THEN
	RETURN;
END_IF
IF xCheck = FALSE THEN
	oldValue := newOrCheckValue;
ELSE
	IF oldValue <> newOrCheckValue THEN
		xTestFailure := TRUE;
	END_IF
END_IF
END_FUNCTION_BLOCK

(* POU Test Bench Folder/TB_SET_REAL, ST *)
FUNCTION_BLOCK TB_SET_REAL
VAR_INPUT
	xEnable: BOOL;
	xCheck: BOOL;
	newOrCheckValue: REAL;
END_VAR
VAR_OUTPUT
	xContinue: BOOL := TRUE;
	xTestFailure: BOOL;
END_VAR
VAR_IN_OUT
	oldValue: REAL;
END_VAR
VAR
END_VAR
IF xEnable = FALSE THEN
	RETURN;
END_IF
IF xCheck = FALSE THEN
	oldValue := newOrCheckValue;
ELSE
	IF oldValue <> newOrCheckValue THEN
		xTestFailure := TRUE;
	END_IF
END_IF
END_FUNCTION_BLOCK

(* POU Test Bench Folder/TB_SET_WORD, ST *)
FUNCTION_BLOCK TB_SET_WORD
VAR_INPUT
	xEnable: BOOL;
	xCheck: BOOL;
	newOrCheckValue: WORD;
END_VAR
VAR_OUTPUT
	xContinue: BOOL := TRUE;
	xTestFailure: BOOL;
END_VAR
VAR_IN_OUT
	oldValue: WORD;
END_VAR
VAR
END_VAR
IF xEnable = FALSE THEN
	RETURN;
END_IF
IF xCheck = FALSE THEN
	oldValue := newOrCheckValue;
ELSE
	IF oldValue <> newOrCheckValue THEN
		xTestFailure := TRUE;
	END_IF
END_IF
END_FUNCTION_BLOCK
